(*

.. <legal notes>

legal notes
=================
| SPDX-FileCopyrightText: © 2026 Oleksandr Tiutyk <trofimich@gmail.com>
| SPDX-License-Identifier: LGPL-3.0-only
| For details check: LGPL-3.0-only_

.. _LGPL-3.0-only: https://www.gnu.org/licenses/lgpl-3.0.en.html

.. </legal notes>

*)

FUNCTION_BLOCK ABSTRACT InputDevice EXTENDS LeafAutomationComponent IMPLEMENTS IInputDevice

METHOD PROTECTED ABSTRACT OnProcessInput
END_METHOD

METHOD FINAL ProcessInput
VAR
	exceptionCode : __SYSTEM.ExceptionCode;
	exception : TOF_Core.IException;
	exceptionReaction : TOF_Core.EXCEPTION_REACTION;
END_VAR
__TRY
	OnProcessInput();
__CATCH(exceptionCode)		
	exception := TOF_Core.ExceptionManager.GetLastException(exceptionCode);
					
	exceptionReaction := OnHandleException(exception, 'OnProcessInput');

	ProcessException(exception, exceptionReaction, "OnProcessInput error");
__ENDTRY
END_METHOD

END_FUNCTION_BLOCK

(* stored: Version 1.1.0.1
   POU InputDevice: Id {efa8b231-2751-492d-8626-738af2170475}, SpecialFunc None
   Folder Methods to override: Id {57e5027c-d025-4d1f-bcea-3cc2ecc52027}
   Method OnProcessInput: Id {30690d44-71d9-48d1-97f7-67db91fa17cb}
   Method ProcessInput: Id {c8983ed6-ea33-4eb7-a3f3-5a36dc5ceb9e} *)
